PROGRAM MAIN
VAR
	getLocalAmsNetId : FB_GetLocalAmsNetId;
	getLocalSystemTime : FB_LocalSystemTime;
	
	id : STRING;
	queryId : STRING;
	stringBuilder : StringBuilder;
	
	original : Bundle;
	confirmed : Bundle;
END_VAR
VAR CONSTANT
	AUTO_RE : INT := 0;
	AUTO_SS : INT := 1;
	MAN_RE : INT := 2;
	MAN_SS : INT := 3;
END_VAR

getLocalSystemTime(
	sNetID:= GVL.AmsNetId, 
	bEnable:= TRUE, 
	dwCycle:= 1, 
	dwOpt:= , 
	tTimeout:= , 
	bValid=> , 
	systemTime=> GVL.systemTime, 
	tzID=> );

IF NOT setup() THEN
	RETURN;
END_IF

MetricMaterialDimensions(GVL.allMaterials);

queryId := stringBuilder
	.concatWith('%')
	.concatWith(id)
	.concatWith('%')
	.getResult();
stringBuilder.reset();

FindBundlesFromDB(id := queryId);

IF confirmed.length <> original.length THEN
	RecalibrateRecipe(original := original, confirmed := confirmed);
	
	IF RecalibrateRecipe.reject THEN //send to manual processes
		confirmed.reqProcesses[AUTO_RE] := FALSE;
		confirmed.reqProcesses[AUTO_SS] := FALSE;
		confirmed.reqProcesses[MAN_RE] := TRUE;
		confirmed.reqProcesses[MAN_SS] := TRUE;	
	END_IF
ELSE
	//use as is
END_IF

METHOD setup : BOOL
VAR_INPUT
END_VAR
getLocalAmsNetId(
	bExecute:= TRUE, 
	tTimeOut:= T#1S, 
	bBusy=> , 
	bError=> , 
	nErrId=> , 
	AddrString=> GVL.AmsNetId, 
	AddrBytes=> );

getLocalAmsNetId.bExecute := FALSE;

setup := (GVL.AmsNetId <> '' AND GVL.AmsNetId <> '0.0.0.0.0.0');
END_METHOD

END_PROGRAM

(* stored: Version 1.1.0.1, ProductVersion 3.1.4024.11
   POU MAIN: Id {2f069ca4-2708-44f0-ace2-897e04b35f3d}, SpecialFunc None
   Method setup: Id {0eefaa89-85b2-413e-a011-eeee3861dbde} *)
